(* IEC 61131-3 sources: plcassist-cli/packages/volt-lsp-iec/test-corpus/pro2193/Device/Plc Logic/Application/99 Library/Function Blocks/Observer Pattern, 7 files *)

(* ---- SubjectBaseFB.fb ---- *)
// A subject is a sensor or button that sends data to attached observers. This base subject does not send any data, only empty events.
{attribute 'no_explicit_call' := 'Do not call this FB. Only use the methods.'}
{attribute 'symbol' := 'none'}
FUNCTION_BLOCK PUBLIC SubjectBaseFB
IMPLEMENTS ISubject, ISubjectBasePayload
VAR
	observers				: ARRAY[1..MaxObservers] OF IObserver;
	{attribute 'hide'}
	_observerCount			: UINT(0..MaxObservers) := 0;
	ui						: UINT;
END_VAR
VAR CONSTANT
	MaxObservers			: UINT := 32;
END_VAR

// More info: https://stefanhenneken.net/2018/05/27/iec-61131-3-the-observer-pattern/

END_FUNCTION_BLOCK

// Attach (subscribe) an observer to this subject. The observer will receive state from the subject.
METHOD PUBLIC Attach : BOOL
VAR_INPUT
	observer			: IObserver;
END_VAR
IF AttachAllowed(observer) THEN
	Attach := AttachObserver(observer);
END_IF
END_METHOD

METHOD PROTECTED AttachAllowed : BOOL
VAR_INPUT
	observer			: IObserver;
END_VAR
VAR
	exclusiveObserver	: IObserverExclusive;
END_VAR
// is the observer NULL?
IF observer = 0 THEN
	LogPlc.Warn('Hey we cannot send messages when observer is NULL!');
	RETURN;
END_IF

// is the observer already registered?
FOR ui := 1 TO ObserverCount DO
	IF observers[ui] = observer THEN
		LogPlc.Warn('Do not attach an observer twice!');
		RETURN;
	END_IF
END_FOR

// are we already attached to an exclusive observer?
IF ObserverCount = 1 AND_THEN __QUERYINTERFACE(observers[1], exclusiveObserver) THEN
	LogPlc.Warn('Use Detach() to remove exclusive observer!');
	DetachAllObservers();
END_IF

// is the new observer Exclusive? If so, detach all observers!
IF __QUERYINTERFACE(observer, exclusiveObserver) THEN
	DetachAllObservers();
END_IF

// is the observer registry full?
IF ObserverCount = MaxObservers THEN
	LogPlc.Fatal('Observer Register Full! Observer will NOT be notified ');
	RETURN;
END_IF

AttachAllowed := TRUE;
END_METHOD

METHOD PROTECTED AttachObserver : BOOL
VAR_INPUT
	observer			: IObserver;
END_VAR
// save the observer object into the array of observers and send the actual value
ObserverCount							:= ObserverCount + 1;
observers[ObserverCount]				:= observer;

// We decided that we do NOT send the current state of the subject when attaching!
//observers[ObserverCount].Update(THIS^);

AttachObserver := TRUE;
END_METHOD

// Detach (unsubscribe) an observer from this subject. The observer do longer receives updates.
METHOD PUBLIC Detach : BOOL
VAR_INPUT
	observer			: IObserver;
END_VAR
VAR
	observerIndex		: UINT;
END_VAR
IF observer = 0 THEN
  RETURN;
END_IF

FOR ui := 1 TO MaxObservers DO
	IF observers[ui] = observer THEN			// Find the observer in the register
		observerIndex := ui;					// Store location where it was found
		observers[ui] := 0;					// Clear the reference
		ObserverCount := ObserverCount - 1;	// Decrease count
		Detach := TRUE;
		EXIT;
	END_IF
END_FOR

IF observerIndex = 0 THEN
	LogPlc.Warn('Detach failed: Observer not found');
END_IF

// Move all references in the register one place up, so there are no gaps in the array.
IF observerIndex > 0 AND observerIndex < MaxObservers THEN
	FOR ui := observerIndex TO MaxObservers - 1 DO
		observers[ui] := observers[ui + 1];
		IF observers[ui + 1] = 0 THEN
			EXIT;
		END_IF
	END_FOR
END_IF
END_METHOD

// Detach (unsubscribe) all observers from this subject.
METHOD PROTECTED DetachAllObservers
FOR ui := 1 TO ObserverCount DO
	observers[ui] := 0;
END_FOR
ObserverCount := 0;
END_METHOD

// Notify all attached observers of state changes
METHOD PUBLIC Notify
FOR ui := 1 TO ObserverCount DO
	observers[ui].Update(THIS^);
END_FOR
END_METHOD

// The actual number of observers that are receiving events
{attribute 'monitoring' := 'call'}
PROPERTY ObserverCount : UINT
GET
VAR
END_VAR
ObserverCount := _observerCount;
END_GET
SET
PROTECTED
VAR
END_VAR
_observerCount := ObserverCount;
END_SET
END_PROPERTY

(* ---- SubjectFunctionKeyFB.fb ---- *)
// A hardware button subject. Send state of HW button to servo drive.
{attribute 'no_explicit_call' := 'Do not call this FB. Only use the methods.'}
{attribute 'hide_all_locals'}
FUNCTION_BLOCK PUBLIC SubjectFunctionKeyFB
EXTENDS SubjectHWButtonFB
IMPLEMENTS ISubject, ISubjectFunctionKeyPayload
VAR
	_extState		: enumFunctionKeyPayload;	// Private backing field for property
END_VAR

END_FUNCTION_BLOCK

// Extended state of the button: tapped, or held, or double-tap-held
{attribute 'monitoring' := 'call'}
PROPERTY ExtState : enumFunctionKeyPayload
GET
VAR
END_VAR
ExtState := _extState;
END_GET
SET
VAR
END_VAR
_extState := ExtState;
END_SET
END_PROPERTY

(* ---- SubjectFunctionKeyFromCodesysVisuFB.fb ---- *)
// A button subject from the CODESYS visu. Has some duplicate code in methods because it overrides logic in SubjectUUIDFB
{attribute 'no_explicit_call' := 'Do not call this FB. Only use the methods.'}
{attribute 'hide_all_locals'}
FUNCTION_BLOCK PUBLIC SubjectFunctionKeyFromCodesysVisuFB
EXTENDS SubjectFunctionKeyFB
IMPLEMENTS ISubject, ISubjectFunctionKeyPayload

END_FUNCTION_BLOCK

// Attach (subscribe) an observer to this subject. The observer will receive state from the subject.
METHOD PUBLIC Attach : BOOL
VAR_INPUT
	observer			: IObserver;
END_VAR

// Code copy from: SubjectBaseFB.Attach()
IF AttachAllowed(observer) THEN
	Attach := AttachObserver(observer);
END_IF
END_METHOD

// Notify all attached observers of state changes
METHOD PUBLIC Notify

// Code copy from: SubjectBaseFB.Notify()
FOR ui := 1 TO ObserverCount DO
	observers[ui].Update(THIS^);
END_FOR
END_METHOD

(* ---- SubjectHWButtonFB.fb ---- *)
// A hardware button subject. Send state of HW button to servo drive.
{attribute 'no_explicit_call' := 'Do not call this FB. Only use the methods.'}
{attribute 'hide_all_locals'}
FUNCTION_BLOCK PUBLIC SubjectHWButtonFB
EXTENDS SubjectUUIDFB
IMPLEMENTS ISubject, ISubjectHWButtonsPayload
VAR
	_buttonType		: enumHWButtons;		// Private backing field for property
	_state			: BOOL;					// Private backing field for property
END_VAR

END_FUNCTION_BLOCK

// Binary state of the button: either pushed or not pushed
{attribute 'monitoring' := 'call'}
PROPERTY ButtonState : BOOL
GET
VAR
END_VAR
ButtonState := _state;
END_GET
SET
VAR
END_VAR
_state := ButtonState;
END_SET
END_PROPERTY

{attribute 'monitoring' := 'call'}
PROPERTY ButtonType : enumHWButtons
GET
VAR
END_VAR
ButtonType := _buttonType;
END_GET
SET
VAR
END_VAR
_buttonType := ButtonType;
END_SET
END_PROPERTY

(* ---- SubjectMouldMeasurementFB.fb ---- *)
// A mould measurement subject.
{attribute 'no_explicit_call' := 'Do not call this FB. Only use the methods.'}
{attribute 'hide_all_locals'}
FUNCTION_BLOCK PUBLIC SubjectMouldMeasurementFB
EXTENDS SubjectBaseFB
IMPLEMENTS ISubject, ISubjectMouldMeasurementPayload
VAR
	_cavity			: INT;							// Private backing field for property
	_classification	: enumMouldMeasurementResult;
	_peakValue		: REAL;
	_shortShotTreshold	: REAL;
END_VAR

END_FUNCTION_BLOCK

{attribute 'monitoring' := 'call'}
PROPERTY Cavity : INT
GET
VAR
END_VAR
Cavity := _cavity;
END_GET
SET

VAR
END_VAR
_cavity := Cavity;
END_SET
END_PROPERTY

PROPERTY Classification : enumMouldMeasurementResult
GET
VAR
END_VAR
Classification := _classification;
END_GET
SET

VAR
END_VAR
_classification := Classification;
END_SET
END_PROPERTY

{attribute 'monitoring' := 'call'}
PROPERTY PeakValue : REAL
GET
VAR
END_VAR
PeakValue := _peakValue;
END_GET
SET

VAR
END_VAR
_peakValue := PeakValue;
END_SET
END_PROPERTY

{attribute 'monitoring' := 'call'}
PROPERTY ShortShotTreshold : REAL
GET
VAR
END_VAR
ShortShotTreshold := _shortShotTreshold;
END_GET
SET

VAR
END_VAR
_shortShotTreshold := ShortShotTreshold;
END_SET
END_PROPERTY

(* ---- SubjectProductionStatisticFB.fb ---- *)
//
{attribute 'no_explicit_call' := 'Do not call this FB. Only use the methods.'}
{attribute 'hide_all_locals'}
{attribute 'symbol' := 'none'}
FUNCTION_BLOCK PUBLIC SubjectProductionStatisticFB
EXTENDS SubjectBaseFB
IMPLEMENTS ISubject, ISubjectProductionStatistic
VAR
	_cavity			: UINT;								// Private backing field for property
	_statType		: enumProductionStatsCavityType;	// Private backing field for property
	_rejectReason	: USINT;							// Private backing field for property
	_data			: UDINT;							// Private backing field for property
END_VAR

END_FUNCTION_BLOCK

// Use like a constructor (kind of) to supply all data to the properties
METHOD PROTECTED NotifyData
VAR_INPUT
	cavity			: UINT;
	statType		: enumProductionStatsCavityType;
	rejectReason	: USINT;
	data			: UDINT;
END_VAR
THIS^.Cavity		:= cavity;
THIS^.StatType		:= statType;
THIS^.RejectReason	:= rejectReason;
THIS^.Data			:= data;

Notify();
END_METHOD

{attribute 'monitoring' := 'call'}
PROPERTY PUBLIC Cavity : UINT
GET
VAR
END_VAR
Cavity := _cavity;
END_GET
SET

VAR
END_VAR
_cavity := Cavity;
END_SET
END_PROPERTY

PROPERTY PUBLIC Data : UDINT
GET
VAR
END_VAR
Data := _data;
END_GET
SET
VAR
END_VAR
_data := Data;
END_SET
END_PROPERTY

PROPERTY PUBLIC RejectReason : USINT
GET
VAR
END_VAR
RejectReason := _rejectReason;
END_GET
SET
VAR
END_VAR
_rejectReason := RejectReason;
END_SET
END_PROPERTY

PROPERTY PUBLIC StatType : enumProductionStatsCavityType
GET
VAR
END_VAR
StatType := _statType;
END_GET
SET

VAR
END_VAR
_statType := StatType;
END_SET
END_PROPERTY

(* ---- SubjectUUIDFB.fb ---- *)
// A special subject that only attaches to observers when a UUID matches
{attribute 'no_explicit_call' := 'Do not call this FB. Only use the methods.'}
FUNCTION_BLOCK PUBLIC SubjectUUIDFB
EXTENDS SubjectBaseFB
IMPLEMENTS ISubject, ISubjectBasePayload
VAR
	storedUUID				: STRING(40);
END_VAR

END_FUNCTION_BLOCK

METHOD PROTECTED AttachAllowed : BOOL
VAR_INPUT
	observer			: IObserver;
END_VAR
IF NOT SUPER^.AttachAllowed(observer) THEN
	AttachAllowed := FALSE;
	RETURN;
END_IF

// There is no manual control screen open, do not allow to connect this observer
IF HMI.UUIDActiveScreen = '' THEN
	LogPlc.Fatal('Trying to attach an observer without a manual control screen open on the HMI');
	AttachAllowed := FALSE;
	RETURN;
END_IF

// is this the first observer to attach to this subject?
IF storedUUID = '' THEN
	storedUUID := HMI.UUIDActiveScreen;
	AttachAllowed := TRUE;
	RETURN;
END_IF

// A new manual control screen was opened. Remove all active observers. Attaching is allowed.
IF storedUUID <> HMI.UUIDActiveScreen THEN
	LogPlc.Warn('Manual control screen on HMI changed without first detaching all observers');
	DetachAllObservers();
	storedUUID := HMI.UUIDActiveScreen;
END_IF

// both UUIDs match, so the new observer is on the same manual control screen. Attaching is allowed.

AttachAllowed := TRUE;
END_METHOD

// Detach (unsubscribe) an observer from this subject. The observer do longer receives updates.
METHOD PUBLIC Detach : BOOL
VAR_INPUT
	observer			: IObserver;
END_VAR
SUPER^.Detach(observer);

IF HMI.UUIDActiveScreen = '' THEN
	storedUUID := '';
END_IF
END_METHOD

METHOD PUBLIC Notify
//Manual control screen was closed or changed, remove all observers!
IF storedUUID <> HMI.UUIDActiveScreen THEN
	IF ObserverCount > 0 THEN
		LogPlc.Warn('Manual control screen on HMI changed, no further action allowed.');
		DetachAllObservers();
	END_IF
	storedUUID := HMI.UUIDActiveScreen;
END_IF

//Only notify observers if any manual control screen is opened on the HMI
IF HMI.UUIDActiveScreen <> '' THEN
	SUPER^.Notify();
END_IF
END_METHOD
